FUNCTION_BLOCK ControlComputation (* Composite Function Block Type *)
  (* Standard: 61499-2 *)
  (* Version 0.0, 2011-12-18, 4DIAC-IDE, 4DIAC-Consortium *)
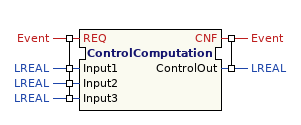
  EVENT_INPUT
    REQ WITH Input1, Input2, Input3; (* Normal Execution Request *)
  END_EVENT
  EVENT_OUTPUT
    CNF WITH ControlOut; (* Execution Confirmation *)
  END_EVENT
  VAR_INPUT
    Input1 : LREAL; (* Input event qualifier *)
    Input2 : LREAL;
    Input3 : LREAL;
  END_VAR
  VAR_OUTPUT
    ControlOut : LREAL; (* Output event qualifier *)
  END_VAR
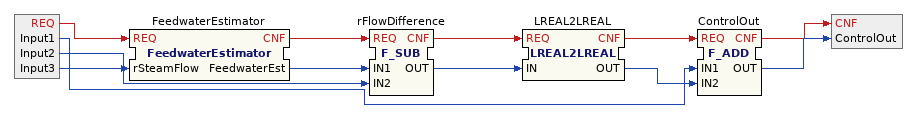
  FBS
    FeedwaterEstimator : FeedwaterEstimator;
    rFlowDifference : F_SUB;
    ControlOut : F_ADD;
    LREAL2LREAL : LREAL2LREAL;
  END_FBS
  EVENT_CONNECTIONS
    REQ TO FeedwaterEstimator.REQ;
    FeedwaterEstimator.CNF TO rFlowDifference.REQ;
    rFlowDifference.CNF TO LREAL2LREAL.REQ;
    LREAL2LREAL.CNF TO ControlOut.REQ;
    ControlOut.CNF TO CNF;
  END_CONNECTIONS
  DATA_CONNECTIONS
    Input3 TO FeedwaterEstimator.rSteamFlow;
    FeedwaterEstimator.FeedwaterEst TO rFlowDifference.IN1;
    Input2 TO rFlowDifference.IN2;
    Input1 TO ControlOut.IN1;
    rFlowDifference.OUT TO LREAL2LREAL.IN;
    LREAL2LREAL.OUT TO ControlOut.IN2;
    ControlOut.OUT TO ControlOut;
  END_CONNECTIONS
END_FUNCTION_BLOCK
